SYSTEM FCCWorkbench
  (* Version 1.0, 2006-08-23, Goran Cengic, Chalmers *)
  DEVICE Test Device : DeviceType_not_used
    RESOURCE Test Resource : ResourceType_not_used
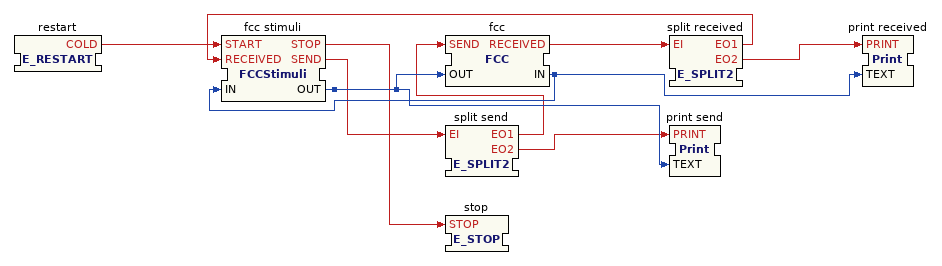
      FBS
        restart : E_RESTART;
        fcc stimuli : FCCStimuli;
        fcc : FCC;
        split send : E_SPLIT2;
        split received : E_SPLIT2;
        print send : Print;
        print received : Print;
        stop : E_STOP;
      END_FBS
      EVENT_CONNECTIONS
        restart.COLD TO fcc stimuli.START;
        fcc stimuli.SEND TO split send.EI;
        split send.EO1 TO fcc.SEND;
        split send.EO2 TO print send.PRINT;
        fcc.RECEIVED TO split received.EI;
        split received.EO1 TO fcc stimuli.RECEIVED;
        split received.EO2 TO print received.PRINT;
        fcc stimuli.STOP TO stop.STOP;
      END_CONNECTIONS
      DATA_CONNECTIONS
        fcc stimuli.OUT TO fcc.OUT;
        fcc.IN TO fcc stimuli.IN;
        fcc stimuli.OUT TO print send.TEXT;
        fcc.IN TO print received.TEXT;
      END_CONNECTIONS
    END_RESOURCE
  END_DEVICE
END_SYSTEM
